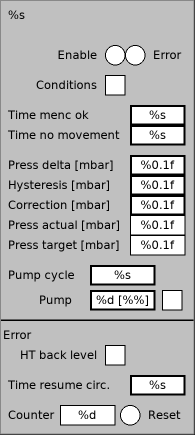
VISUALIZATION _VISU_InkCirculation  // 195x435
VAR_IN_OUT
  m_Inst_Fb : FB_InkCirculation;               (*visu fb instance*) 
END_VAR
    Rectangle (0,0 195x320)
    Rectangle (5,5 180x20), "%s", text variable: m_Inst_Fb._sName
    Ellipse (105,45 20x20), colour toggle: m_Inst_Fb.IbEnable
        toggle m_Inst_Fb.IbEnable
    Rectangle (10,45 90x20), "Enable"
    Ellipse (125,45 20x20), colour toggle: m_Inst_Fb.bLevelError, invisible if: NOT m_Inst_Fb.bLevelError
        toggle m_Inst_Fb.bLevelError
    Rectangle (150,45 40x20), "Error", invisible if: NOT m_Inst_Fb.bLevelError
    Rectangle (5,155 120x20), "Press delta [mbar]"
    Rectangle (130,155 55x20), "%0.1f", text variable: m_Inst_Fb.fRSubMencDeltaP
        OnMouseDown: write the text variable via Edit, min -20, max 0
    Rectangle (5,215 120x20), "Press actual [mbar]"
    Rectangle (130,215 55x20), "%0.1f", text variable: m_Inst_Fb.fSubMencActValue
    Rectangle (5,235 120x20), "Press target [mbar]"
    Rectangle (130,235 55x20), "%0.1f", text variable: m_Inst_Fb.fSubMencTargetValue
    RoundedRectangle (162,290 20x20), colour toggle: m_Inst_Fb.bPumpActivation
    Rectangle (25,290 50x20), "Pump"
    RoundedRectangle (105,75 20x20), colour toggle: m_Inst_Fb.bConditionsMet
    Rectangle (10,75 90x20), "Conditions"
    Rectangle (5,175 120x20), "Hysteresis [mbar]"
    Rectangle (130,175 55x20), "%0.1f", text variable: m_Inst_Fb.fRSubMencHysteresisP
        OnMouseDown: write the text variable via Edit, min 0, max 5
    Rectangle (5,105 120x20), "Time menc ok"
    Rectangle (130,105 55x20), "%s", text variable: m_Inst_Fb.tRSubMencOk
        OnMouseDown: write the text variable via Edit
    Rectangle (5,125 120x20), "Time no movement"
    Rectangle (130,125 55x20), "%s", text variable: m_Inst_Fb.tRNoMovement
        OnMouseDown: write the text variable via Edit
    Rectangle (0,320 195x115)
    Rectangle (0,325 90x20), "Error"
    RoundedRectangle (105,345 20x20), colour toggle: m_Inst_Fb.IbInkLevelReachedBack
    Rectangle (10,345 90x20), "HT back level"
    Rectangle (5,375 120x20), "Time resume circ."
    Rectangle (130,375 55x20), "%s", text variable: m_Inst_Fb.tRResumeCirculation
        OnMouseDown: write the text variable via Edit
    Rectangle (5,405 60x20), "Counter"
    Rectangle (60,405 55x20), "%d", text variable: m_Inst_Fb.nRErrorCounter
    Ellipse (120,405 20x20)
        tap m_Inst_Fb.bResetErrorCounter
    Rectangle (145,405 45x20), "Reset"
    Rectangle (5,195 120x20), "Correction [mbar]"
    Rectangle (130,195 55x20), "%0.1f", text variable: m_Inst_Fb.fRSubMencCorrectionP
        OnMouseDown: write the text variable via Edit, min -1, max 1
    Rectangle (5,265 80x20), "Pump cycle"
    Rectangle (90,265 65x20), "%s", text variable: m_Inst_Fb.tRPumpDutyCycleFrequency
        OnMouseDown: write the text variable via Edit
    Rectangle (90,290 65x20), "%d [%%]", text variable: m_Inst_Fb.nRPumpDutyCycle
        OnMouseDown: write the text variable via Edit
END_VISUALIZATION

(* stored: Version 1.1.0.1, ProductVersion 3.1.4024.11
   Visu _VISU_InkCirculation: Id {22cb4460-f6b0-4f31-acce-18c5125256e4} *)
